Yaskawa INFORM job: SKRZYNIA_4840_0_STOPNI_1OBR.JBI

/JOB
//NAME SKRZYNIA_4840_0_STOPNI_1OBR
///FOLDERNAME 02-SKRZYNIE_JOBS
//POS
///NPOS 505,505,0,43,0,0
///TOOL 0
///POSTYPE PULSE
///PULSE
C00000=1055,-24125,84372,288,19725,204
C00001=1055,-24125,84372,288,19725,204
C00002=0,-15438,65714,0,-68532,0
C00003=25524,-25821,36823,19654,-58495,38520
C00004=23988,-24960,37134,18595,-57837,38812
C00005=22822,-23954,37534,17811,-57199,39017
C00006=22935,-24057,37491,17887,-57262,38997
C00007=20006,-24258,37408,15644,-56932,39751
C00008=24402,-25289,37013,18874,-58060,38740
C00009=22585,-24665,40358,17164,-59622,30036
C00010=23477,-23257,40205,18030,-58646,29630
C00011=22519,-22398,40568,17384,-58125,29795
C00012=22700,-22567,40495,17506,-58225,29764
C00013=19339,-22794,40398,14955,-57865,30607
C00014=24825,-24328,39798,18931,-59350,29401
C00015=32755,-32613,25711,29640,-48730,33694
C00016=25632,-30899,26166,23992,-46203,35378
C00017=24264,-29862,26497,22996,-45413,35639
C00018=24403,-29974,26459,23097,-45496,35612
C00019=20575,-30233,26374,19602,-44891,36810
C00020=26556,-31526,25988,24663,-46720,35206
C00021=30467,-39837,7164,47016,-28378,22959
C00022=27667,-31817,21023,40298,-29340,25942
C00023=26226,-30681,21430,39338,-28403,26129
C00024=26403,-30829,21375,39455,-28520,26106
C00025=23300,-31093,21277,35654,-27590,27434
C00026=27667,-31817,21023,40298,-29340,25942
C00027=26028,-43665,26580,-39946,8682,24640
C00028=27956,-30595,53065,-101898,6609,54413
C00029=26028,-43663,26580,-39944,8677,24639
C00030=38124,-35330,25507,26155,-45940,34419
C00031=17528,-33021,25719,14295,-44761,40001
C00032=28412,-21339,35361,20830,-70681,36412
C00033=27333,-20260,35973,20228,-70115,36596
C00034=27560,-20497,35837,20355,-70235,36556
C00035=24830,-20816,35654,18694,-69859,37222
C00036=28877,-18893,40191,20941,-72149,36569
C00037=27817,-32566,25782,25532,-47502,36865
C00038=25779,-31294,26110,24054,-46400,37243
C00039=24344,-30243,26427,23007,-45578,37515
C00040=24432,-30312,26405,23072,-45630,37498
C00041=20021,-30599,26315,19050,-44944,38872
C00042=26262,-31616,26021,24405,-46667,37153
C00043=27439,-32346,25835,25259,-47302,36935
C00044=25659,-31170,26146,23974,-46312,37260
C00045=24581,-30384,26384,23190,-45695,37464
C00046=24689,-30466,26358,23269,-45758,37444
C00047=20001,-30771,26264,18999,-45026,38899
C00048=26308,-31607,26026,24448,-46671,37139
C00049=29920,-29398,24569,49034,-27892,27689
C00050=29115,-28721,24834,48649,-27358,27707
C00051=27674,-27540,25333,47889,-26423,27783
C00052=27794,-27645,25287,47952,-26502,27777
C00053=24751,-27949,25156,44290,-25406,29014
C00054=29115,-28721,24834,48649,-27358,27707
C00055=46709,-36638,22429,58955,-37174,26391
C00056=28781,-29734,22128,31822,13650,18140
C00057=28781,-29734,22128,31822,47214,18140
C00058=28781,-29734,22128,31822,47214,18140
C00059=54276,-43673,-470,62120,-47739,23626
C00060=41752,-40945,238,55421,-40682,25053
C00061=39867,-39951,547,54583,-39468,25162
C00062=39963,-40004,529,54625,-39531,25157
C00063=37168,-40414,400,52318,-38319,25966
C00064=43368,-42081,-2849,57747,-40820,23950
C00065=38095,-40136,7813,41252,-44156,24924
C00066=33231,-38681,8176,37792,-41757,25918
C00067=31538,-37640,8473,36716,-40716,26179
C00068=31687,-37737,8444,36811,-40809,26155
C00069=27389,-38154,8322,32773,-39589,27627
C00070=33834,-39023,8084,38175,-42120,25821
C00071=27585,-47842,-289,32095,-40789,28095
C00072=4801,-35772,25187,4593,-28023,-82032
C00073=17634,-23800,39238,9573,-31425,-73339
C00074=17634,-23800,39238,9573,-31425,-73339
C00075=16549,-22464,39800,8390,-30730,-72975
C00076=16684,-22641,39722,8536,-30818,-73021
C00077=16684,-19968,45512,8078,-32771,-72767
C00078=17634,-23800,39238,9573,-31425,-73339
C00079=17837,-21535,44509,9322,-33342,-73155
C00080=17837,-21535,44509,9322,-33342,-73155
C00081=16866,-20378,45014,8305,-32755,-72853
C00082=17032,-20588,44918,8481,-32857,-72905
C00083=17032,-17542,51480,8009,-35060,-72636
C00084=17837,-21535,44509,9322,-33342,-73155
C00085=-20829,-18800,50532,-12466,-37179,-77446
C00086=-19934,-17904,50946,-11618,-36715,-77676
C00087=-20044,-18019,50891,-11723,-36773,-77647
C00088=-20044,-15288,56753,-11218,-38713,-77950
C00089=-20966,-18928,50473,-12596,-37250,-77413
C00090=-20884,-26676,33664,-14451,-31668,-76336
C00091=-20884,-26676,33664,-14451,-31668,-76336
C00092=-19557,-25338,34176,-13080,-30873,-76751
C00093=-19691,-25483,34117,-13220,-30955,-76709
C00094=-19691,-22773,39998,-12506,-32911,-77106
C00095=-20642,-26447,33747,-14206,-31526,-76411
C00096=-33629,-40566,17444,-29603,-33447,-71192
C00097=-33629,-40566,17444,42578,-32312,-84654
C00098=-42160,-31266,16400,42578,-32312,-84654
C00099=-87798,-804,48829,-20188,-26072,-60966
C00100=-76454,-11934,10236,-25964,7954,-64922
C00101=-76448,-11928,10235,-25961,7944,-64914
C00102=-68643,-7759,-23318,-14097,50582,-74897
C00103=-70868,-8793,-8075,-29663,30364,-70765
C00104=-67243,-1968,12282,-49553,26687,-63567
C00105=-68655,-309,14069,-48513,25966,-64203
C00106=-67497,-1678,12591,-49367,26558,-63682
C00107=-71436,-723,2905,-26484,35140,-73726
C00108=-71436,176,6426,-27636,33595,-73066
C00109=-71434,778,8668,-28412,32633,-72624
C00110=-68624,-2689,-85,-28291,36551,-72622
C00111=-99375,3692,5712,40719,48607,-84097
C00112=-94964,4957,10918,40408,44640,-83792
C00113=-93063,6047,12199,39572,43744,-83178
C00114=-94964,4957,10918,40408,44640,-83792
C00115=-94964,5754,13918,41385,43553,-84439
C00116=-94964,4957,10918,40408,44640,-83792
C00117=-90271,-412,-5146,23417,46876,-76529
C00118=-83133,-4088,-8267,6704,41492,-71542
C00119=-83133,-4088,-8267,6704,41492,-71542
C00120=-83133,-4088,-8267,6704,41492,-11598
C00121=-83133,-16026,-8267,6704,41492,-11598
C00122=-83133,-16026,-8267,6704,41492,-11598
C00123=-48225,-19387,30619,3889,32460,-6728
C00124=56943,-39861,25115,1795,-37402,-69601
C00125=29960,-38386,-19607,-115769,-41858,-24264
C00126=65721,-6478,18155,-133323,-22195,3361
C00127=70544,4411,32968,-134868,-18623,4660
C00128=71874,8263,38598,-134556,-17327,4659
C00129=72629,9390,40002,-135279,-16924,5107
C00130=71441,7638,37831,-134139,-17555,4406
C00131=77146,8888,25050,-166574,-32612,18372
C00132=77146,10029,28643,-166204,-31014,18167
C00133=77146,11198,32202,-165803,-29459,17947
C00134=75508,4678,16951,-165715,-35157,17778
C00135=68680,12216,24468,-164340,-40455,-13359
C00136=68362,12845,25743,-164045,-40097,-13561
C00137=68362,13700,28585,-163752,-38808,-13742
C00138=68362,12845,25743,-164045,-40097,-13561
C00139=64993,-1168,28876,-102971,-10760,-49875
C00140=63888,481,30670,-102324,-11438,-50313
C00141=64993,-1168,28876,-102971,-10760,-49875
C00142=58588,-14653,4620,-120782,-19611,-35794
C00143=29960,-38386,-19607,-115769,-41858,-24264
C00144=56943,-39861,25115,1795,-37402,-69601
C00145=-1002,-39861,25115,1795,-37402,-69601
C00146=-1001,-39858,25114,1795,-37402,0
C00147=6591,-33902,35532,5956,-1761,-1932
C00148=6592,-33900,35531,103508,-35512,-26314
C00149=-99253,-13690,44082,59847,13407,-31313
C00150=-85045,-36869,-4353,28502,-22832,-52282
C00151=-92346,-18713,13565,21110,-22545,-55257
C00152=-85732,-21202,11427,30682,-24763,-59235
C00153=-84559,-15616,15722,33768,-24118,-60665
C00154=-84150,-13282,17685,34842,-23935,-61163
C00155=-83260,-12880,18034,36130,-24218,-61709
C00156=-84150,-13282,17685,34842,-23935,-61163
C00157=-85365,-11775,19006,33430,-23307,-60600
C00158=-84150,-13282,17685,34842,-23935,-61163
C00159=-85786,-16909,14677,31743,-23900,-59790
C00160=-84150,-13282,17685,34842,-23935,-61163
C00161=-83215,-12861,18051,36194,-24233,-61735
C00162=-84150,-13282,17685,34842,-23935,-61163
C00163=-85327,-11825,18959,33476,-23327,-60618
C00164=-84150,-13282,17685,34842,-23935,-61163
C00165=-87841,-18519,13420,28367,-23534,-58339
C00166=-84150,-13282,17685,34842,-23935,-61163
C00167=-83292,-12894,18020,36083,-24208,-61688
C00168=-84150,-13282,17685,34842,-23935,-61163
C00169=-85185,-12008,18799,33646,-23400,-60687
C00170=-84150,-13282,17685,34842,-23935,-61163
C00171=-86371,-18277,13606,30568,-23951,-59265
C00172=-84345,-13370,17612,34554,-23873,-61041
C00173=-83240,-12871,18042,36158,-24225,-61720
C00174=-84345,-13370,17612,34554,-23873,-61041
C00175=-85365,-12110,18711,33368,-23345,-60568
C00176=-84345,-13370,17612,34554,-23873,-61041
C00177=-86191,-19647,12567,30467,-24278,-59187
C00178=-84345,-13372,17610,34552,-23873,-61039
C00179=-83096,-12807,18098,36363,-24268,-61804
C00180=-84345,-13372,17610,34552,-23873,-61039
C00181=-85268,-12232,18600,33480,-23393,-60612
C00182=-84345,-13372,17610,34552,-23873,-61039
C00183=-84814,-16043,15376,33312,-24093,-60464
C00184=-84104,-13265,17702,34906,-23948,-61189
C00185=-82960,-12743,18153,36555,-24313,-61887
C00186=-84104,-13265,17702,34906,-23948,-61189
C00187=-84979,-12194,18635,33901,-23496,-60788
C00188=-84104,-13265,17702,34906,-23948,-61189
C00189=-86610,-16845,14732,30573,-23614,-59301
C00190=-84104,-13265,17702,34906,-23948,-61189
C00191=-82793,-12667,18222,36790,-24370,-61986
C00192=-84104,-13265,17702,34906,-23948,-61189
C00193=-84888,-12305,18537,34004,-23540,-60830
C00194=-84104,-13265,17702,34906,-23948,-61189
C00195=-83806,-19585,12613,33764,-25080,-60559
C00196=-83675,-13072,17868,35530,-24083,-61453
C00197=-82553,-12556,18319,37130,-24451,-62127
C00198=-83675,-13072,17868,35530,-24083,-61453
C00199=-84378,-12223,18610,34735,-23716,-61138
C00200=-83675,-13072,17868,35530,-24083,-61453
C00201=-87149,-17993,13826,29513,-23647,-58830
C00202=-84104,-13265,17702,34906,-23948,-61189
C00203=-82640,-12594,18285,37014,-24425,-62079
C00204=-84104,-13265,17702,34906,-23948,-61189
C00205=-84792,-12429,18430,34119,-23592,-60877
C00206=-84104,-13265,17702,34906,-23948,-61189
C00207=-83583,-9185,30892,23668,-36042,-57025
C00208=-85789,-8328,35795,20592,-37093,-55378
C00209=-85786,-16735,14816,31782,-23869,-59812
C00210=-84103,-13263,17702,34906,-23947,-61191
C00211=-83225,-12865,18046,36177,-24227,-61729
C00212=-84103,-13263,17702,34906,-23947,-61191
C00213=-84774,-12447,18412,34138,-23599,-60886
C00214=-84103,-13263,17702,34906,-23947,-61191
C00215=-86149,-16246,6730,18897,-35239,-57128
C00216=-86244,-15289,7532,18875,-35060,-57127
C00217=-85361,-14893,7870,19824,-35193,-57574
C00218=-86244,-15289,7532,18875,-35060,-57127
C00219=-86889,-14409,8282,18264,-34784,-56850
C00220=-86244,-15289,7532,18875,-35060,-57127
C00221=-90262,-21765,2389,14114,-35574,-54847
C00222=-90262,-21765,2389,28730,-17672,-54847
C00223=-89967,-19086,25635,28730,-17672,-54847
C00224=568,-24029,84339,168,19981,112
C00225=568,-24677,83015,164,20405,113
C00226=101153,-24598,83176,165,20353,113
C00227=101153,-24598,83176,165,20353,113
C00228=89967,-19086,25635,-28730,-17672,54847
C00229=90262,-21765,2389,-28730,-17672,54847
C00230=86932,-18662,4771,-17876,-35519,56628
C00231=86578,-15436,7408,-18515,-35011,56957
C00232=85428,-14922,7844,-19753,-35183,57541
C00233=84405,-14447,8250,-20842,-35348,58054
C00234=85428,-14922,7844,-19753,-35183,57541
C00235=86134,-13973,8661,-19091,-34881,57237
C00236=85428,-14922,7844,-19753,-35183,57541
C00237=85786,-16735,14816,-31782,-23869,59812
C00238=83514,-12996,17929,-35760,-24132,61552
C00239=82296,-12429,18424,-37488,-24534,62281
C00240=83514,-12996,17929,-35760,-24132,61552
C00241=84266,-12085,18725,-34910,-23738,61214
C00242=83514,-12996,17929,-35760,-24132,61552
C00243=87323,-6914,39851,-18853,-38149,44508
C00244=83118,-12818,18089,-36330,-24263,61791
C00245=81969,-12276,18566,-37944,-24648,62472
C00246=83118,-12818,18089,-36330,-24263,61791
C00247=83927,-11846,18941,-35423,-23842,61433
C00248=83118,-12818,18089,-36330,-24263,61791
C00249=83806,-19585,12613,-33764,-25080,60559
C00250=83148,-12832,18077,-36287,-24254,61773
C00251=81889,-12236,18598,-38058,-24676,62520
C00252=83148,-12832,18077,-36287,-24254,61773
C00253=83900,-11930,18867,-35446,-23862,61440
C00254=83148,-12832,18077,-36287,-24254,61773
C00255=86610,-16845,14732,-30573,-23614,59301
C00256=82493,-13239,17725,-37070,-24559,62089
C00257=81442,-12739,18159,-38529,-24915,62703
C00258=82493,-13239,17725,-37070,-24559,62089
C00259=83435,-12133,18689,-36040,-24063,61682
C00260=82493,-13239,17725,-37070,-24559,62089
C00261=84814,-16043,15376,-33312,-24093,60464
C00262=82555,-13613,17404,-36910,-24580,62015
C00263=81369,-13053,17885,-38558,-24979,62709
C00264=82555,-13613,17404,-36910,-24580,62015
C00265=83568,-12431,18429,-35805,-24046,61580
C00266=82555,-13613,17404,-36910,-24580,62015
C00267=86191,-19647,12567,-30467,-24278,59187
C00268=82500,-13648,17375,-36975,-24607,62039
C00269=81594,-13224,17740,-38236,-24911,62571
C00270=82500,-13648,17375,-36975,-24607,62039
C00271=83449,-12543,18332,-35941,-24104,61633
C00272=82500,-13648,17375,-36975,-24607,62039
C00273=86371,-18277,13606,-30568,-23951,59265
C00274=82904,-13790,17251,-36416,-24470,61808
C00275=81796,-13275,17692,-37971,-24838,62464
C00276=82904,-13790,17251,-36416,-24470,61808
C00277=83696,-12867,18046,-35547,-24051,61466
C00278=82904,-13790,17251,-36416,-24470,61808
C00279=87841,-18519,13420,-28367,-23534,58339
C00280=82748,-13879,17174,-36603,-24542,61883
C00281=81789,-13434,17554,-37946,-24861,62449
C00282=82748,-13879,17174,-36603,-24542,61883
C00283=83603,-12888,18026,-35668,-24086,61514
C00284=82748,-13879,17174,-36603,-24542,61883
C00285=85786,-16909,14677,-31743,-23900,59790
C00286=82339,-14116,16972,-37087,-24733,62079
C00287=81557,-13752,17280,-38171,-24994,62536
C00288=82339,-14116,16972,-37087,-24733,62079
C00289=83390,-12909,18006,-35951,-24172,61633
C00290=82339,-14116,16972,-37087,-24733,62079
C00291=85732,-21202,11427,-30682,-24763,59235
C00292=82398,-14365,16763,-36952,-24745,62014
C00293=81340,-13876,17176,-38416,-25096,62632
C00294=82398,-14365,16763,-36952,-24745,62014
C00295=83629,-12951,17972,-35620,-24090,61491
C00296=82398,-14365,16763,-36952,-24745,62014
C00297=83775,-36460,5778,-32556,-23750,56951
C00298=69856,-53931,-13446,-33557,-28911,29591
C00299=0,-24029,84339,0,19981,0
C00300=0,-24029,84339,0,19981,0
C00301=0,-52280,40443,0,6876,0
C00302=43695,-41610,22646,45477,-37580,9181
C00303=79833,-32060,29151,65065,-75499,17030
C00304=46589,-23543,32575,47437,-59456,19719
C00305=35046,-28601,21000,31995,-60106,26294
C00306=20995,-31929,9410,15929,-60729,34224
C00307=58029,-25484,23838,55879,-68285,17494
C00308=64424,-28491,31029,58630,-66351,17656
C00309=0,-52280,40443,0,6876,0
C00310=0,-52280,40443,0,6876,0
C00311=23755,-47704,18289,26329,-25233,13971
C00312=32804,-46073,6525,41905,-31120,14425
C00313=62562,-39100,6547,70046,-55853,12125
C00314=48126,-33841,8393,64372,-47199,12361
C00315=31253,-44096,-7366,36514,-42480,22085
C00316=59828,-44646,-5405,72855,-48572,12139
C00317=0,-38761,66314,0,-763,0
C00318=0,-44757,54667,0,2744,0
C00319=40382,-38226,12225,48505,-40693,16039
C00320=55481,-27484,23768,62968,-54833,11978
C00321=49931,-26522,24223,59987,-51967,12537
C00322=41382,-34078,10932,46059,-50502,16311
C00323=55330,-33748,11238,57660,-59334,12681
C00324=78664,-24436,10378,82837,-79111,12029
C00325=75189,-23065,11287,81851,-76948,11927
C00326=75189,-45249,11287,81851,-38847,11927
C00327=29880,-45249,11287,43145,-11324,11927
C00328=0,-24029,84339,0,19981,0
C00329=0,-24026,84338,1,19977,2
C00330=4264,-34194,25387,4006,-26954,-29436
C00331=4264,-34194,25387,4006,-26954,-81856
C00332=-21478,-27798,32214,-15234,-31599,-76056
C00333=-19679,-23059,39354,-12567,-32689,-77067
C00334=16724,-20576,44291,8212,-32395,-72836
C00335=21329,-26386,39716,13285,-34016,-74401
C00336=-23778,-26243,38799,-16502,-35132,-75964
C00337=-20075,-15782,55752,-11329,-38404,-77896
C00338=16874,-17447,51356,7863,-34895,-72604
C00339=18580,-28601,30698,11472,-29284,-74138
C00340=6126,-41331,18955,6697,-26557,-30383
C00341=1,-24024,84337,2,19973,1
C00342=-64243,-26178,31107,-39513,40312,-5844
C00343=-72148,3973,56008,-35470,42045,-10522
C00344=-72090,16396,76301,-42067,35650,-6519
C00345=-69388,15725,61378,-31740,35177,-8719
C00346=-69127,27099,75569,-32744,34250,-8088
C00347=-67573,2495,11285,-21767,57629,-15193
C00348=-77819,19629,29798,-10454,63174,-20704
C00349=-72990,23583,14304,-10735,77209,-20379
C00350=-74593,38003,46707,-11043,65751,-19814
C00351=-73236,38943,48295,-11400,65557,-19316
C00352=-73329,42107,51779,-6346,67443,-19636
C00353=-87142,34654,46174,17622,63862,-25393
C00354=-87240,36727,48611,18897,66604,-25032
C00355=-99033,21517,12213,24947,79702,-26203
C00356=-91500,-14196,-34781,24472,81625,-22832
C00357=-100472,-45007,-27818,8167,67201,-29302
C00358=0,-36642,16905,0,48372,0
C00359=66009,-61997,-62105,21406,63483,18379
C00360=97242,-23579,-39442,10179,68876,30321
C00361=73684,-7073,-17511,24638,68131,29022
C00362=59136,7235,6676,33270,66602,27507
C00363=54816,14937,6234,39741,69494,31070
C00364=54365,20668,19279,41017,66202,29418
C00365=64503,4223,2857,29650,48528,26647
C00366=75622,3202,-3149,3890,49494,34281
C00367=88036,13177,2413,-18568,66573,35876
C00368=90462,21593,10123,-22613,76266,34479
C00369=92450,29224,20002,-25750,81642,33727
C00370=94949,8131,-12163,-20291,74229,36861
C00371=94949,8084,-13484,-20215,75047,36712
C00372=70412,-34016,-52305,-11724,65624,29757
C00373=44268,-30306,-1568,-7370,48673,18708
C00374=1,-24024,84337,2,19973,1
C00375=1,-24024,84337,2,19973,1
C00376=3796,-57671,22373,2336,-25309,-753
C00377=52632,-34554,16626,51161,-63050,5622
C00378=41454,-25301,37199,36495,-58855,24340
C00379=36675,-26014,30916,36565,-54296,30358
C00380=27394,-45680,-17645,86603,-20054,2054
C00381=62932,-33588,12189,66848,-61063,18031
C00382=55769,-31640,17107,64026,-54372,11197
C00383=49968,-26926,23568,59773,-52215,12586
C00384=49609,-31413,12230,55051,-55993,13121
C00385=55330,-33748,11238,57660,-59334,12681
C00386=29694,-28537,50295,31543,-18263,8508
C00387=1,-24024,84337,2,19973,1
C00388=1,-24024,84337,2,19973,1
C00389=57188,-41777,19973,48132,-58706,4905
C00390=55566,-48748,-16991,79805,-45048,-6941
C00391=49908,-48716,-25784,90749,-41340,-3650
C00392=34097,-50090,-26426,85195,-27377,-3312
C00393=25337,-51401,-46092,139691,-32480,-30357
C00394=55456,-69347,-61742,105381,-46819,-11205
C00395=12119,-24859,71505,13236,4440,2633
C00396=-91085,-34291,10385,1908,-24348,-42097
C00397=-86191,-19647,12567,30467,-24278,-59187
C00398=-99336,-11722,19052,-14323,-20229,-40037
C00399=-98356,-11562,19564,-10422,-20330,-41507
C00400=-99474,-20389,12397,-11593,-22150,-41069
C00401=0,-52280,40443,0,6876,0
C00402=98750,-34911,19055,13387,-20552,33529
C00403=85481,-22689,10385,-30594,-25183,59147
C00404=97204,-12655,18233,8807,-19987,42423
C00405=97248,-12883,18033,8874,-20029,42393
C00406=96230,-24528,9149,6144,-22576,43630
C00407=0,-52280,40443,0,6876,0
C00408=0,-52280,40443,0,6876,0
C00409=-90140,-60305,18108,-2708,1721,-7625
C00410=-95594,-27428,6866,-4663,-19832,-42154
C00411=-99356,-13410,18355,-15385,-17730,-37479
C00412=-99591,-10931,20459,-16242,-17374,-37088
C00413=-99412,-10883,20509,-15863,-17339,-37249
C00414=-100555,-16348,15834,-17428,-18409,-36628
C00415=-90140,-60305,18108,-2708,1721,-7625
C00416=0,-52280,40443,0,6876,0
C00417=84259,-57935,27522,-3761,3673,6310
C00418=86507,-39672,4297,-27618,-16640,46340
C00419=79502,-31038,5321,-35142,-29552,60614
C00420=87509,-17632,14108,-29072,-23467,58651
C00421=100494,-12641,18246,19637,-20925,37756
C00422=99867,-15453,10402,24266,-14765,33998
C00423=100699,-20865,6123,24471,-16015,33991
C00424=86507,-39672,4297,-27618,-16640,46340
C00425=84259,-57935,27522,-3761,3673,6310
C00426=0,-52280,40443,0,6876,0
C00427=0,-27933,77061,0,20812,0
C00428=0,-27933,77061,0,20812,0
C00429=0,-52280,40443,0,6876,0
C00430=-91970,-60791,14435,-3343,512,-9412
C00431=-99196,-15868,16098,-13748,-19297,-38710
C00432=-99196,-15868,16098,-13748,-19297,-38710
C00433=-99196,-15868,16098,-13748,-19297,-38710
C00434=-85896,-11794,19566,31613,-21074,-58206
C00435=-87494,-11929,19445,26784,-20178,-56163
C00436=-99562,-16264,15781,-14410,-19427,-38431
C00437=-99196,-15868,16098,-13748,-19297,-38710
C00438=-91970,-60791,14435,-3343,512,-9412
C00439=0,-52280,40443,0,6876,0
C00440=91083,-60784,14823,-9043,-825,15173
C00441=83869,-19403,12921,-33769,-24740,60260
C00442=83869,-19403,12921,-33769,-24740,60260
C00443=83420,-14897,16486,-35538,-24144,61113
C00444=90681,-11839,19658,-13770,-20778,51433
C00445=90505,-11641,19895,-14005,-20849,51502
C00446=95871,-14889,15992,4901,-19605,43825
C00447=83869,-19403,12921,-33769,-24740,60260
C00448=91083,-60784,14823,-9043,-825,15173
C00449=0,-52280,40443,0,6876,0
C00450=-91526,-60598,16699,7584,176,-13289
C00451=-94392,-6553,48683,5805,-47321,-49764
C00452=-88951,-345,54953,10686,-47392,-51569
C00453=-88305,5764,62037,11205,-47732,-51744
C00454=-91201,-14114,9416,8552,-34389,-51801
C00455=-84917,-15593,15742,33275,-23984,-60461
C00456=-81669,-15982,15425,37506,-25258,-62202
C00457=-79867,-25377,9541,37586,-25936,-59971
C00458=-91415,-60262,16631,7870,-73,-13734
C00459=24,-24029,84339,7,19981,5
C00460=160,-24029,84339,47,19981,32
C00461=99096,-24029,84339,47,19981,32
C00462=99096,-24029,84339,47,19981,32
C00463=89967,-19086,25635,-28730,-17672,54847
C00464=85786,-16735,14816,-31782,-23869,59812
C00465=83492,-14473,16674,-35480,-24338,61406
C00466=82747,-11488,19289,-37317,-24361,62210
C00467=85506,-13730,8787,-19466,-34817,57474
C00468=85505,-16299,6686,-19564,-35388,57437
C00469=89967,-19086,25635,-28730,-17672,54847
C00470=568,-24029,84339,168,19981,112
C00471=568,-24029,84339,168,19981,112
C00472=-91970,-60791,14435,-3343,512,-9412
C00473=-86948,-23217,10819,28314,-23349,-56438
C00474=-85895,-16522,15767,31843,-22281,-58087
C00475=-93744,1669,52928,2829,-38206,-34736
C00476=-93484,-766,47198,3260,-36104,-34933
C00477=-86145,-24679,9854,29028,-23971,-56682
C00478=-100471,-58311,4157,14142,-4822,-27614
C00479=-68517,-58311,4157,14142,-4822,-27614
C00480=0,-52280,40443,0,6876,0
C00481=91083,-60784,14823,-9043,-825,15173
C00482=83869,-19403,12921,-33769,-24740,60260
C00483=82620,-18743,14708,-32942,-26226,58979
C00484=84031,-4887,35984,-19530,-40379,54984
C00485=84316,-7987,27276,-19995,-38113,55712
C00486=84798,-22668,11879,-29033,-26372,57255
C00487=91083,-60784,14823,-9043,-825,15173
C00488=0,-52280,40443,0,6876,0
C00489=-6369,-39206,65423,-4801,-482,2563
C00490=-97287,-29142,12714,-8673,-22288,-37832
C00491=-86191,-19647,12567,30467,-24278,-59187
C00492=-85671,-16302,15857,30808,-24404,-58999
C00493=-100216,-10426,22391,-15020,-22581,-38655
C00494=-96259,-10424,22189,-2878,-17380,-43087
C00495=-87910,-17792,15835,25414,-24996,-56048
C00496=-97287,-29142,12714,-8673,-22288,-37832
C00497=0,-52280,40443,0,6876,0
C00498=92301,-25634,22749,2368,-15645,37646
C00499=83738,-18329,13570,-34202,-24868,60772
C00500=90255,-12942,18284,-15153,-20833,52586
C00501=93508,-13158,18002,-4292,-20124,47959
C00502=80226,-20465,12178,-39626,-27411,62762
C00503=92301,-25634,22749,2368,-15645,37646
C00504=0,-52280,40443,0,6876,0
BC00000=413138
BC00001=413138
BC00002=413138
BC00003=413134
BC00004=413134
BC00005=413134
BC00006=413134
BC00007=413134
BC00008=413134
BC00009=474623
BC00010=474628
BC00011=474628
BC00012=474628
BC00013=474628
BC00014=474628
BC00015=522849
BC00016=522849
BC00017=522849
BC00018=522849
BC00019=522849
BC00020=522849
BC00021=550624
BC00022=544410
BC00023=544410
BC00024=544410
BC00025=544410
BC00026=544410
BC00027=461029
BC00028=618860
BC00029=673957
BC00030=691345
BC00031=686969
BC00032=712250
BC00033=712250
BC00034=712250
BC00035=712250
BC00036=712250
BC00037=708270
BC00038=708270
BC00039=708270
BC00040=708270
BC00041=708270
BC00042=708270
BC00043=770184
BC00044=770184
BC00045=770184
BC00046=770184
BC00047=770184
BC00048=770184
BC00049=779519
BC00050=779519
BC00051=779519
BC00052=779519
BC00053=779519
BC00054=779519
BC00055=720678
BC00056=703565
BC00057=703565
BC00058=802913
BC00059=891475
BC00060=891475
BC00061=891475
BC00062=891475
BC00063=891475
BC00064=891475
BC00065=919114
BC00066=919114
BC00067=919114
BC00068=919114
BC00069=919114
BC00070=919114
BC00071=919114
BC00072=865069
BC00073=880430
BC00074=880430
BC00075=880430
BC00076=880430
BC00077=880430
BC00078=880430
BC00079=884876
BC00080=884876
BC00081=884876
BC00082=884876
BC00083=884876
BC00084=884876
BC00085=884876
BC00086=884876
BC00087=884876
BC00088=884876
BC00089=884876
BC00090=884876
BC00091=884876
BC00092=884876
BC00093=884876
BC00094=884876
BC00095=884876
BC00096=884876
BC00097=884876
BC00098=884876
BC00099=884876
BC00100=884876
BC00101=902628
BC00102=913714
BC00103=930418
BC00104=930418
BC00105=930418
BC00106=930418
BC00107=930418
BC00108=930418
BC00109=930419
BC00110=930419
BC00111=930419
BC00112=930419
BC00113=930419
BC00114=930419
BC00115=930419
BC00116=930419
BC00117=920796
BC00118=906162
BC00119=880897
BC00120=880897
BC00121=880897
BC00122=847715
BC00123=813282
BC00124=884876
BC00125=884876
BC00126=884876
BC00127=901090
BC00128=906251
BC00129=906251
BC00130=906251
BC00131=906251
BC00132=906251
BC00133=906251
BC00134=906251
BC00135=906251
BC00136=906251
BC00137=906251
BC00138=906251
BC00139=906251
BC00140=906251
BC00141=906251
BC00142=900738
BC00143=854154
BC00144=838793
BC00145=838793
BC00146=854156
BC00147=785093
BC00148=785096
BC00149=785096
BC00150=854699
BC00151=886829
BC00152=902188
BC00153=902188
BC00154=902188
BC00155=902188
BC00156=902188
BC00157=902188
BC00158=902188
BC00159=840744
BC00160=840744
BC00161=840744
BC00162=840744
BC00163=840744
BC00164=840744
BC00165=779300
BC00166=779300
BC00167=779300
BC00168=779300
BC00169=779300
BC00170=779300
BC00171=717855
BC00172=717855
BC00173=717855
BC00174=717855
BC00175=717855
BC00176=717855
BC00177=656405
BC00178=656405
BC00179=656405
BC00180=656405
BC00181=656405
BC00182=656405
BC00183=594961
BC00184=594961
BC00185=594961
BC00186=594961
BC00187=594961
BC00188=594961
BC00189=533517
BC00190=533517
BC00191=533517
BC00192=533517
BC00193=533517
BC00194=533517
BC00195=472073
BC00196=472073
BC00197=472073
BC00198=472073
BC00199=472073
BC00200=472073
BC00201=410629
BC00202=410629
BC00203=410629
BC00204=410629
BC00205=410629
BC00206=410629
BC00207=410629
BC00208=349186
BC00209=349186
BC00210=349186
BC00211=349186
BC00212=349186
BC00213=349186
BC00214=349186
BC00215=336469
BC00216=336469
BC00217=336469
BC00218=336469
BC00219=336469
BC00220=336469
BC00221=336469
BC00222=336469
BC00223=336469
BC00224=336469
BC00225=511557
BC00226=512005
BC00227=363797
BC00228=336469
BC00229=336469
BC00230=337415
BC00231=337415
BC00232=337415
BC00233=337415
BC00234=337415
BC00235=337415
BC00236=337415
BC00237=349186
BC00238=350137
BC00239=350137
BC00240=350137
BC00241=350137
BC00242=350137
BC00243=410629
BC00244=411580
BC00245=411580
BC00246=411580
BC00247=411580
BC00248=411580
BC00249=472073
BC00250=473025
BC00251=473025
BC00252=473025
BC00253=473025
BC00254=473025
BC00255=533517
BC00256=534468
BC00257=534468
BC00258=534468
BC00259=534468
BC00260=534468
BC00261=594961
BC00262=594961
BC00263=594961
BC00264=594961
BC00265=594961
BC00266=594961
BC00267=656405
BC00268=657350
BC00269=657350
BC00270=657350
BC00271=657350
BC00272=657350
BC00273=717855
BC00274=718799
BC00275=718799
BC00276=718799
BC00277=718799
BC00278=718799
BC00279=779300
BC00280=780245
BC00281=780245
BC00282=780245
BC00283=780245
BC00284=780245
BC00285=840744
BC00286=841691
BC00287=841691
BC00288=841691
BC00289=841691
BC00290=841691
BC00291=902188
BC00292=903136
BC00293=903136
BC00294=903136
BC00295=903136
BC00296=903136
BC00297=866428
BC00298=742376
BC00299=673191
BC00300=769966
BC00301=716865
BC00302=723595
BC00303=717171
BC00304=717171
BC00305=716481
BC00306=715784
BC00307=716000
BC00308=727625
BC00309=716865
BC00310=820009
BC00311=882789
BC00312=908954
BC00313=917484
BC00314=918947
BC00315=923719
BC00316=887066
BC00317=801718
BC00318=476098
BC00319=466373
BC00320=456696
BC00321=456696
BC00322=417276
BC00323=417276
BC00324=493986
BC00325=514306
BC00326=485368
BC00327=469222
BC00328=459569
BC00329=774064
BC00330=862181
BC00331=867397
BC00332=884876
BC00333=884876
BC00334=880429
BC00335=874663
BC00336=870174
BC00337=884876
BC00338=884876
BC00339=884104
BC00340=887696
BC00341=735557
BC00342=750919
BC00343=750919
BC00344=807629
BC00345=827515
BC00346=852454
BC00347=884386
BC00348=884386
BC00349=911895
BC00350=911895
BC00351=911895
BC00352=911896
BC00353=911896
BC00354=911897
BC00355=911897
BC00356=911897
BC00357=826555
BC00358=785153
BC00359=868693
BC00360=907813
BC00361=907814
BC00362=907814
BC00363=938061
BC00364=938061
BC00365=938061
BC00366=938061
BC00367=938061
BC00368=938064
BC00369=938064
BC00370=938064
BC00371=911658
BC00372=911658
BC00373=842845
BC00374=735557
BC00375=469153
BC00376=499904
BC00377=541592
BC00378=531564
BC00379=529848
BC00380=571759
BC00381=529848
BC00382=333808
BC00383=332068
BC00384=295166
BC00385=294388
BC00386=454783
BC00387=441730
BC00388=632615
BC00389=778314
BC00390=778312
BC00391=778312
BC00392=778312
BC00393=826760
BC00394=836556
BC00395=566410
BC00396=707357
BC00397=656405
BC00398=656405
BC00399=717855
BC00400=717855
BC00401=680147
BC00402=662303
BC00403=657350
BC00404=657350
BC00405=718803
BC00406=718803
BC00407=683493
BC00408=792672
BC00409=792672
BC00410=896850
BC00411=895720
BC00412=895720
BC00413=925351
BC00414=927080
BC00415=792672
BC00416=792672
BC00417=792672
BC00418=887446
BC00419=903126
BC00420=903126
BC00421=903126
BC00422=936389
BC00423=936389
BC00424=887446
BC00425=792672
BC00426=792672
BC00427=700249
BC00428=546214
BC00429=546214
BC00430=546211
BC00431=546211
BC00432=406776
BC00433=406776
BC00434=406778
BC00435=468200
BC00436=468200
BC00437=546211
BC00438=546211
BC00439=546214
BC00440=546214
BC00441=507604
BC00442=410782
BC00443=410782
BC00444=410782
BC00445=472720
BC00446=472720
BC00447=507604
BC00448=546214
BC00449=546214
BC00450=516757
BC00451=383716
BC00452=349186
BC00453=349186
BC00454=336469
BC00455=349186
BC00456=410629
BC00457=416512
BC00458=515801
BC00459=520018
BC00460=474013
BC00461=474013
BC00462=403108
BC00463=336469
BC00464=349186
BC00465=349186
BC00466=349186
BC00467=337415
BC00468=337415
BC00469=336469
BC00470=336469
BC00471=428401
BC00472=546211
BC00473=591088
BC00474=591088
BC00475=591088
BC00476=531116
BC00477=529640
BC00478=529640
BC00479=529640
BC00480=529640
BC00481=546214
BC00482=589919
BC00483=595627
BC00484=609761
BC00485=555903
BC00486=534177
BC00487=546214
BC00488=529640
BC00489=651195
BC00490=765890
BC00491=777968
BC00492=778453
BC00493=779252
BC00494=832733
BC00495=840748
BC00496=730002
BC00497=671551
BC00498=714120
BC00499=780224
BC00500=780222
BC00501=841743
BC00502=841743
BC00503=741100
BC00504=660586
///POSTYPE BASE
///RECTAN
///RCONF 1,0,0,0,0,0,0,0,0,0,0,0,0,0,0,0,0,0,0,0,0,0,0,0
P00006=0.000,0.000,0.000,0.0000,0.0000,0.0000
///RCONF 0,0,0,0,0,0,0,0,0,0,0,0,0,0,0,0,0,0,0,0,0,0,0,0
P00021=6.550,-0.003,-5.735,0.0000,0.0000,0.0000
P00022=5.943,-0.018,-6.388,0.0000,0.0000,0.0000
P00023=7.025,-0.019,-7.168,0.0000,0.0000,0.0000
P00024=5.926,-0.047,-4.777,0.0000,0.0000,0.0000
///RCONF 1,0,0,0,0,0,0,0,0,0,0,0,0,0,0,0,0,0,0,0,0,0,0,0
P00098=-0.089,-2.467,4.059,0.0000,0.0000,0.0000
P00099=0.011,-2.380,1.226,0.0000,0.0000,0.0000
P00100=-0.081,2.558,4.482,0.0000,0.0000,0.0000
P00101=0.030,-2.286,2.993,0.0000,0.0000,0.0000
P00102=-0.005,-1.108,1.644,0.0000,0.0000,0.0000
P00103=-0.094,-3.400,4.200,0.0000,0.0000,0.0000
P00104=0.043,-2.127,5.826,0.0000,0.0000,0.0000
P00105=-0.043,0.662,5.286,0.0000,0.0000,0.0000
P00106=-0.018,-2.519,0.237,0.0000,0.0000,0.0000
P00107=-0.008,-4.537,-4.500,0.0000,0.0000,0.0000
P00108=0.014,-3.040,2.637,0.0000,0.0000,0.0000
P00109=0.017,-3.622,2.341,0.0000,0.0000,0.0000
///RCONF 0,0,0,0,0,0,0,0,0,0,0,0,0,0,0,0,0,0,0,0,0,0,0,0
P00280=-0.761,-1.221,0.004,0.0000,0.0000,0.0000
///RCONF 1,0,0,0,0,0,0,0,0,0,0,0,0,0,0,0,0,0,0,0,0,0,0,0
P00281=-0.866,-3.587,-0.008,0.0000,0.0000,0.0000
///RCONF 0,0,0,0,1,0,0,0,0,0,0,0,0,0,0,0,0,0,0,0,0,0,0,0
P00290=-0.023,-0.050,5.560,0.0000,0.0000,0.0000
///RCONF 1,0,0,0,0,0,0,0,0,0,0,0,0,0,0,0,0,0,0,0,0,0,0,0
P00291=0.002,-0.893,4.526,0.0000,0.0000,0.0000
P00301=0.046,-2.112,7.779,0.0000,0.0000,0.0000
P00302=-0.180,-2.409,6.326,0.0000,0.0000,0.0000
///RCONF 0,0,0,0,0,0,0,0,0,0,0,0,0,0,0,0,0,0,0,0,0,0,0,0
P00303=-0.004,-1.437,-4.584,0.0000,0.0000,0.0000
P00304=0.028,-1.666,-4.234,0.0000,0.0000,0.0000
P00305=-0.003,-1.920,-3.501,0.0000,0.0000,0.0000
P00306=0.015,-2.252,-3.054,0.0000,0.0000,0.0000
P00307=0.019,-2.151,-5.077,0.0000,0.0000,0.0000
P00308=-0.003,-2.092,-4.888,0.0000,0.0000,0.0000
P00309=-0.040,-2.205,-4.992,0.0000,0.0000,0.0000
P00310=-0.006,-2.490,-5.925,0.0000,0.0000,0.0000
P00311=-0.007,-2.079,-5.307,0.0000,0.0000,0.0000
P00350=11.519,-0.008,1.149,0.0000,0.0000,0.0000
P00351=13.563,-0.027,-0.653,0.0000,0.0000,0.0000
P00352=13.252,-0.027,-0.827,0.0000,0.0000,0.0000
P00353=10.971,-0.082,0.776,0.0000,0.0000,0.0000
P00354=-0.024,2.508,-1.824,0.0000,0.0000,0.0000
P00355=-0.001,2.528,-1.131,0.0000,0.0000,0.0000
P00356=-0.034,2.921,-0.262,0.0000,0.0000,0.0000
P00357=0.003,3.386,-0.091,0.0000,0.0000,0.0000
P00358=0.014,3.037,-0.020,0.0000,0.0000,0.0000
P00359=-0.005,2.731,0.912,0.0000,0.0000,0.0000
P00360=-0.011,3.412,0.438,0.0000,0.0000,0.0000
//INST
///DATE 2025/06/04 08:15
///ATTR SC,RW
///GROUP1 RB1,BS1
NOP
CALL JOB:MOVE_INTO_TUNNEL
MOVJ C00000 BC00000 VJ=30.00
'------------------------
'------------------------
'SPOINA SRODEK DOL
'------------------------
'------------------------
'POMIAR DO WYJ!! PRZEROBIC NA STD
MOVJ C00001 BC00001 VJ=40.00
MOVJ C00002 BC00002 VJ=40.00
'W3P
MOVJ C00003 BC00003 VJ=20.00 PL=0
MOVL C00004 BC00004 V=166.7 PL=0
REFP 3 C00005 BC00005
CALL JOB:SEARCH-R1
SET P0100 P0006
SFTON P0100
MOVL C00006 BC00006 V=66.7 PL=0
REFP 3 C00007 BC00007
CALL JOB:SEARCH-R1
SET P0100 P0006
SFTON P0100
MOVL C00008 BC00008 V=333.3 PL=0
SFTOF
'W3L
MOVL C00009 BC00009 V=666.7
MOVL C00010 BC00010 V=166.7 PL=0
REFP 3 C00011 BC00011
CALL JOB:SEARCH-R1
SET P0101 P0006
SFTON P0101
MOVL C00012 BC00012 V=166.7 PL=0
REFP 3 C00013 BC00013
CALL JOB:SEARCH-R1
SET P0101 P0006
SFTON P0101
MOVL C00014 BC00014 V=333.3 PL=0
SFTOF
'W9P
MOVL C00015 BC00015 V=666.7
MOVL C00016 BC00016 V=166.7
REFP 3 C00017 BC00017
CALL JOB:SEARCH-R1
SET P0102 P0006
SFTON P0102
MOVL C00018 BC00018 V=166.7 PL=0
REFP 3 C00019 BC00019
CALL JOB:SEARCH-R1
SET P0102 P0006
SFTON P0102
SFTOF
MOVL C00020 BC00020 V=333.3 PL=0
'W9L
MOVL C00021 BC00021 V=666.7
MOVL C00022 BC00022 V=166.7
REFP 3 C00023 BC00023
CALL JOB:SEARCH-R1
SET P0103 P0006
SFTON P0103
MOVL C00024 BC00024 V=166.7 PL=0
REFP 3 C00025 BC00025
CALL JOB:SEARCH-R1
SET P0103 P0006
SFTON P0103
MOVL C00026 BC00026 V=333.3 PL=0
SFTOF
'PRZEJAZ NAD BELKA
MOVL C00027 BC00027 V=666.7
MOVJ C00028 BC00028 VJ=40.00
MOVJ C00029 BC00029 VJ=40.00
MOVJ C00030 BC00030 VJ=40.00
'W1P
SFTOF
MOVJ C00031 BC00031 VJ=20.00 PL=0
MOVL C00032 BC00032 V=166.7 PL=0
REFP 3 C00033 BC00033
CALL JOB:SEARCH-R1
SET P0104 P0006
SFTON P0104
MOVL C00034 BC00034 V=166.7 PL=0
REFP 3 C00035 BC00035
CALL JOB:SEARCH-R1
SET P0104 P0006
SFTON P0104
MOVL C00036 BC00036 V=333.3 PL=0
SFTOF
'W1L
MOVL C00037 BC00037 V=666.7
MOVL C00038 BC00038 V=166.7 PL=0
REFP 3 C00039 BC00039
CALL JOB:SEARCH-R1
SET P0105 P0006
SFTON P0105
MOVL C00040 BC00040 V=166.7 PL=0
REFP 3 C00041 BC00041
CALL JOB:SEARCH-R1
SET P0105 P0006
SFTON P0105
MOVL C00042 BC00042 V=333.3 PL=0
SFTOF
MOVL C00043 BC00043 V=666.7
'W10P
MOVL C00044 BC00044 V=166.7 PL=0
REFP 3 C00045 BC00045
CALL JOB:SEARCH-R1
SET P0106 P0006
SFTON P0106
MOVL C00046 BC00046 V=166.7 PL=0
REFP 3 C00047 BC00047
CALL JOB:SEARCH-R1
SET P0106 P0006
SFTON P0106
MOVL C00048 BC00048 V=333.3 PL=0
SFTOF
'W10L
MOVL C00049 BC00049 V=333.3
MOVL C00050 BC00050 V=166.7 PL=0
REFP 3 C00051 BC00051
CALL JOB:SEARCH-R1
SET P0107 P0006
SFTON P0107
MOVL C00052 BC00052 V=166.7 PL=0
REFP 3 C00053 BC00053
CALL JOB:SEARCH-R1
SET P0107 P0006
SFTON P0107
MOVL C00054 BC00054 V=333.3 PL=0
SFTOF
MOVL C00055 BC00055 V=333.3
MOVL C00056 BC00056 V=333.3
MOVL C00057 BC00057 V=333.3
MOVL C00058 BC00058 V=833.3
MOVL C00059 BC00059 V=333.3
MOVL C00060 BC00060 V=166.7 PL=0
REFP 3 C00061 BC00061
CALL JOB:SEARCH-R1
SET P0108 P0006
SFTON P0108
MOVL C00062 BC00062 V=166.7 PL=0
REFP 3 C00063 BC00063
CALL JOB:SEARCH-R1
SET P0108 P0006
SFTON P0108
MOVL C00064 BC00064 V=333.3 PL=0
SFTOF
'PRZEJAZD
MOVL C00065 BC00065 V=666.7
MOVL C00066 BC00066 V=166.7 PL=0
REFP 3 C00067 BC00067
CALL JOB:SEARCH-R1
SET P0109 P0006
SFTON P0109
MOVL C00068 BC00068 V=166.7 PL=0
REFP 3 C00069 BC00069
CALL JOB:SEARCH-R1
SET P0109 P0006
SFTON P0109
MOVL C00070 BC00070 V=333.3 PL=0
SFTOF
'PRZEJAZD
'POMIAR DO WYJ!! PRZEROBIC NA STD
'KONIEC
MOVJ C00071 BC00071 VJ=25.00
MOVJ C00072 BC00072 VJ=50.00
'W5L
MOVJ C00073 BC00073 VJ=30.00 PL=0
MOVL C00074 BC00074 V=166.7
REFP 3 C00075 BC00075
CALL JOB:SEARCH-R1
SET P0021 P0006
SFTON P0021
MOVL C00076 BC00076 V=166.7
REFP 3 C00077 BC00077
CALL JOB:SEARCH-R1
SET P0021 P0006
SFTON P0021
SFTOF
MOVL C00078 BC00078 V=166.7
'W6L
MOVJ C00079 BC00079 VJ=20.00 PL=0
MOVL C00080 BC00080 V=166.7
REFP 3 C00081 BC00081
CALL JOB:SEARCH-R1
SET P0022 P0006
SFTON P0022
MOVL C00082 BC00082 V=166.7
REFP 3 C00083 BC00083
CALL JOB:SEARCH-R1
SET P0022 P0006
SFTON P0022
SFTOF
MOVL C00084 BC00084 V=166.7
'W6P
MOVL C00085 BC00085 V=333.3 PL=0
REFP 3 C00086 BC00086
CALL JOB:SEARCH-R1
SET P0023 P0006
SFTON P0023
MOVL C00087 BC00087 V=166.7
REFP 3 C00088 BC00088
CALL JOB:SEARCH-R1
SET P0023 P0006
SFTON P0023
SFTOF
MOVL C00089 BC00089 V=166.7
'W5P
MOVJ C00090 BC00090 VJ=20.00 PL=0
MOVL C00091 BC00091 V=166.7
REFP 3 C00092 BC00092
CALL JOB:SEARCH-R1
SET P0024 P0006
SFTON P0024
MOVL C00093 BC00093 V=166.7
REFP 3 C00094 BC00094
CALL JOB:SEARCH-R1
SET P0024 P0006
SFTON P0024
SFTOF
MOVL C00095 BC00095 V=166.7
'W7A
MOVJ C00096 BC00096 VJ=40.00
MOVJ C00097 BC00097 VJ=40.00
MOVJ C00098 BC00098 VJ=40.00
MOVJ C00099 BC00099 VJ=40.00
MOVJ C00100 BC00100 VJ=40.00
MOVJ C00101 BC00101 VJ=40.00
MOVJ C00102 BC00102 VJ=40.00
MOVJ C00103 BC00103 VJ=40.00
MOVL C00104 BC00104 V=250.0
REFP 3 C00105 BC00105
CALL JOB:SEARCH-R1
SET P0280 P0006
SFTON P0280
MOVL C00106 BC00106 V=166.7
MOVL C00107 BC00107 V=250.0
MOVL C00108 BC00108 V=166.7
REFP 3 C00109 BC00109
CALL JOB:SEARCH-R1
SET P0280 P0006
MOVL C00110 BC00110 V=166.7
SFTOF
MOVL C00111 BC00111 V=333.3
MOVL C00112 BC00112 V=166.7
REFP 3 C00113 BC00113
CALL JOB:SEARCH-R1
SET P0290 P0006
SFTON P0290
MOVL C00114 BC00114 V=166.7
REFP 3 C00115 BC00115
CALL JOB:SEARCH-R1
SET P0290 P0006
MOVL C00116 BC00116 V=166.7
'DOKONCZYC SEARCH
'DOKONCZYC SEARCH
MOVJ C00117 BC00117 VJ=20.00
SFTOF
MOVJ C00118 BC00118 VJ=30.00
MOVJ C00119 BC00119 VJ=40.00
MOVJ C00120 BC00120 VJ=40.00
MOVJ C00121 BC00121 VJ=40.00
MOVJ C00122 BC00122 VJ=40.00
MOVJ C00123 BC00123 VJ=50.00
'W7B
MOVJ C00124 BC00124 VJ=50.00
MOVJ C00125 BC00125 VJ=50.00
MOVJ C00126 BC00126 VJ=30.00
MOVJ C00127 BC00127 VJ=20.00
MOVL C00128 BC00128 V=166.7
REFP 3 C00129 BC00129
CALL JOB:SEARCH-R1
SET P0281 P0006
MOVL C00130 BC00130 V=166.7
SFTON P0281
MOVL C00131 BC00131 V=166.7
MOVL C00132 BC00132 V=166.7
REFP 3 C00133 BC00133
CALL JOB:SEARCH-R1
SET P0281 P0006
MOVJ C00134 BC00134 VJ=15.00
SFTOF
MOVJ C00135 BC00135 VJ=20.00
MOVL C00136 BC00136 V=166.7
REFP 3 C00137 BC00137
CALL JOB:SEARCH-R1
SET P0291 P0006
MOVL C00138 BC00138 V=166.7
MOVL C00139 BC00139 V=166.7
REFP 3 C00140 BC00140
CALL JOB:SEARCH-R1
SET P0291 P0006
MOVL C00141 BC00141 V=166.7
MOVJ C00142 BC00142 VJ=30.00
MOVJ C00143 BC00143 VJ=30.00
MOVJ C00144 BC00144 VJ=50.00
MOVJ C00145 BC00145 VJ=50.00
'------------------------
'------------------------
'PRAWA STRONA PROFIL GORA
'------------------------
'------------------------
MOVJ C00146 BC00146 VJ=50.00
MOVJ C00147 BC00147 VJ=50.00
MOVJ C00148 BC00148 VJ=50.00
MOVJ C00149 BC00149 VJ=20.00
MOVJ C00150 BC00150 VJ=50.00
'------------------------
'W14A L
'------------------------
SFTOF
MOVJ C00151 BC00151 VJ=50.00
'------------------------
'W14A P
'------------------------
SFTOF
MOVJ C00152 BC00152 VJ=50.00
MOVJ C00153 BC00153 VJ=50.00
MOVL C00154 BC00154 V=166.7 PL=0
REFP 3 C00155 BC00155
CALL JOB:SEARCH-R1
SET P0301 P0006
SFTON P0301
MOVL C00156 BC00156 V=166.7 PL=0
REFP 3 C00157 BC00157
CALL JOB:SEARCH-R1
SET P0301 P0006
SFTON P0301
MOVL C00158 BC00158 V=166.7 PL=0
SFTOF
'------------------------
'W19A L
'------------------------
SFTOF
MOVJ C00159 BC00159 VJ=50.00
MOVL C00160 BC00160 V=200.0 PL=0
REFP 3 C00161 BC00161
CALL JOB:SEARCH-R1
SET P0302 P0006
SFTON P0302
MOVL C00162 BC00162 V=166.7 PL=0
REFP 3 C00163 BC00163
CALL JOB:SEARCH-R1
SET P0302 P0006
SFTON P0302
MOVL C00164 BC00164 V=250.0 PL=0
SFTOF
'------------------------
'W19A P
'------------------------
SFTOF
MOVJ C00165 BC00165 VJ=50.00
MOVL C00166 BC00166 V=166.7 PL=0
REFP 3 C00167 BC00167
CALL JOB:SEARCH-R1
SET P0303 P0006
SFTON P0303
MOVL C00168 BC00168 V=166.7 PL=0
REFP 3 C00169 BC00169
CALL JOB:SEARCH-R1
SET P0303 P0006
SFTON P0303
MOVL C00170 BC00170 V=166.7 PL=0
SFTOF
'------------------------
'W13A L
'------------------------
SFTOF
MOVJ C00171 BC00171 VJ=50.00
MOVL C00172 BC00172 V=166.7 PL=0
REFP 3 C00173 BC00173
CALL JOB:SEARCH-R1
SET P0304 P0006
SFTON P0304
MOVL C00174 BC00174 V=166.7 PL=0
REFP 3 C00175 BC00175
CALL JOB:SEARCH-R1
SET P0304 P0006
SFTON P0304
MOVL C00176 BC00176 V=166.7 PL=0
SFTOF
'------------------------
'W13A P
'------------------------
SFTOF
MOVJ C00177 BC00177 VJ=50.00
MOVL C00178 BC00178 V=200.0 PL=0
REFP 3 C00179 BC00179
CALL JOB:SEARCH-R1
SET P0305 P0006
SFTON P0305
MOVL C00180 BC00180 V=166.7 PL=0
REFP 3 C00181 BC00181
CALL JOB:SEARCH-R1
SET P0305 P0006
SFTON P0305
MOVL C00182 BC00182 V=250.0 PL=0
SFTOF
'------------------------
'W18A L
'------------------------
SFTOF
MOVJ C00183 BC00183 VJ=50.00
MOVL C00184 BC00184 V=200.0 PL=0
REFP 3 C00185 BC00185
CALL JOB:SEARCH-R1
SET P0306 P0006
SFTON P0306
MOVL C00186 BC00186 V=166.7 PL=0
REFP 3 C00187 BC00187
CALL JOB:SEARCH-R1
SET P0306 P0006
SFTON P0306
MOVL C00188 BC00188 V=166.7 PL=0
SFTOF
'------------------------
'W18A P
'------------------------
SFTOF
MOVJ C00189 BC00189 VJ=50.00
MOVL C00190 BC00190 V=200.0 PL=0
REFP 3 C00191 BC00191
CALL JOB:SEARCH-R1
SET P0307 P0006
SFTON P0307
MOVL C00192 BC00192 V=166.7 PL=0
REFP 3 C00193 BC00193
CALL JOB:SEARCH-R1
SET P0307 P0006
SFTON P0307
MOVL C00194 BC00194 V=166.7 PL=0
SFTOF
'------------------------
'W15A L
'------------------------
SFTOF
MOVJ C00195 BC00195 VJ=50.00
MOVL C00196 BC00196 V=200.0 PL=0
REFP 3 C00197 BC00197
CALL JOB:SEARCH-R1
SET P0308 P0006
SFTON P0308
MOVL C00198 BC00198 V=166.7 PL=0
REFP 3 C00199 BC00199
CALL JOB:SEARCH-R1
SET P0308 P0006
SFTON P0308
MOVL C00200 BC00200 V=166.7 PL=0
SFTOF
'------------------------
'W15A P
'------------------------
SFTOF
MOVJ C00201 BC00201 VJ=50.00
MOVL C00202 BC00202 V=166.7 PL=0
REFP 3 C00203 BC00203
CALL JOB:SEARCH-R1
SET P0309 P0006
SFTON P0309
MOVL C00204 BC00204 V=166.7 PL=0
REFP 3 C00205 BC00205
CALL JOB:SEARCH-R1
SET P0309 P0006
SFTON P0309
MOVL C00206 BC00206 V=166.7 PL=0
SFTOF
MOVL C00207 BC00207 V=333.3
'------------------------
'W17A L
'------------------------
MOVL C00208 BC00208 V=500.0
SFTOF
MOVJ C00209 BC00209 VJ=20.00
MOVL C00210 BC00210 V=166.7 PL=0
REFP 3 C00211 BC00211
CALL JOB:SEARCH-R1
SET P0310 P0006
SFTON P0310
MOVL C00212 BC00212 V=166.7 PL=0
REFP 3 C00213 BC00213
CALL JOB:SEARCH-R1
SET P0310 P0006
SFTON P0310
MOVL C00214 BC00214 V=166.7 PL=0
SFTOF
'------------------------
'W17A P
'------------------------
SFTOF
MOVL C00215 BC00215 V=416.7
MOVL C00216 BC00216 V=166.7 PL=0
REFP 3 C00217 BC00217
CALL JOB:SEARCH-R1
SET P0311 P0006
SFTON P0311
MOVL C00218 BC00218 V=166.7 PL=0
REFP 3 C00219 BC00219
CALL JOB:SEARCH-R1
SET P0311 P0006
SFTON P0311
MOVL C00220 BC00220 V=166.7 PL=0
SFTOF
MOVJ C00221 BC00221 VJ=10.00
MOVJ C00222 BC00222 VJ=20.00
MOVJ C00223 BC00223 VJ=50.00
MOVJ C00224 BC00224 VJ=50.00
MOVJ C00225 BC00225 VJ=70.00
MOVJ C00226 BC00226 VJ=30.00
MOVJ C00227 BC00227 VJ=30.00
'------------------------
'------------------------
'LEWA STRONA PROFIL GORA
'------------------------
'------------------------
MOVJ C00228 BC00228 VJ=30.00
MOVJ C00229 BC00229 VJ=30.00
MOVJ C00230 BC00230 VJ=30.00
'------------------------
'W17B L
'------------------------
SFTOF
MOVJ C00231 BC00231 VJ=15.00
MOVL C00232 BC00232 V=166.7 PL=0
REFP 3 C00233 BC00233
CALL JOB:SEARCH-R1
SET P0350 P0006
SFTON P0350
MOVL C00234 BC00234 V=166.7 PL=0
REFP 3 C00235 BC00235
CALL JOB:SEARCH-R1
SET P0350 P0006
SFTON P0350
MOVL C00236 BC00236 V=166.7 PL=0
SFTOF
'------------------------
'W17B P
'------------------------
SFTOF
MOVL C00237 BC00237 V=333.3
MOVL C00238 BC00238 V=166.7 PL=0
REFP 3 C00239 BC00239
CALL JOB:SEARCH-R1
SET P0351 P0006
SFTON P0351
MOVL C00240 BC00240 V=166.7 PL=0
REFP 3 C00241 BC00241
CALL JOB:SEARCH-R1
SET P0351 P0006
SFTON P0351
MOVL C00242 BC00242 V=166.7 PL=0
SFTOF
'POPRAWID DOJAZD
'------------------------
'W15B L
'------------------------
SFTOF
MOVJ C00243 BC00243 VJ=10.00
MOVL C00244 BC00244 V=166.7 PL=0
REFP 3 C00245 BC00245
CALL JOB:SEARCH-R1
SET P0352 P0006
SFTON P0352
MOVL C00246 BC00246 V=166.7 PL=0
REFP 3 C00247 BC00247
CALL JOB:SEARCH-R1
SET P0352 P0006
SFTON P0352
MOVL C00248 BC00248 V=166.7 PL=0
SFTOF
'------------------------
'W15B P
'------------------------
SFTOF
MOVJ C00249 BC00249 VJ=20.00
MOVL C00250 BC00250 V=166.7 PL=0
REFP 3 C00251 BC00251
CALL JOB:SEARCH-R1
SET P0353 P0006
SFTON P0353
MOVL C00252 BC00252 V=166.7 PL=0
REFP 3 C00253 BC00253
CALL JOB:SEARCH-R1
SET P0353 P0006
SFTON P0353
MOVL C00254 BC00254 V=166.7 PL=0
SFTOF
'------------------------
'W18B L
'------------------------
SFTOF
MOVJ C00255 BC00255 VJ=50.00
MOVL C00256 BC00256 V=166.7 PL=0
REFP 3 C00257 BC00257
CALL JOB:SEARCH-R1
SET P0354 P0006
SFTON P0354
MOVL C00258 BC00258 V=166.7 PL=0
REFP 3 C00259 BC00259
CALL JOB:SEARCH-R1
SET P0354 P0006
SFTON P0354
MOVL C00260 BC00260 V=166.7 PL=0
SFTOF
'------------------------
'W18B P
'------------------------
SFTOF
MOVJ C00261 BC00261 VJ=50.00
MOVL C00262 BC00262 V=166.7 PL=0
REFP 3 C00263 BC00263
CALL JOB:SEARCH-R1
SET P0355 P0006
SFTON P0355
MOVL C00264 BC00264 V=166.7 PL=0
REFP 3 C00265 BC00265
CALL JOB:SEARCH-R1
SET P0355 P0006
SFTON P0355
MOVL C00266 BC00266 V=166.7 PL=0
SFTOF
'------------------------
'W13B L
'------------------------
SFTOF
MOVJ C00267 BC00267 VJ=50.00
MOVL C00268 BC00268 V=166.7 PL=0
REFP 3 C00269 BC00269
CALL JOB:SEARCH-R1
SET P0356 P0006
SFTON P0356
MOVL C00270 BC00270 V=166.7 PL=0
REFP 3 C00271 BC00271
CALL JOB:SEARCH-R1
SET P0356 P0006
SFTON P0356
MOVL C00272 BC00272 V=166.7 PL=0
SFTOF
'------------------------
'W13B P
'------------------------
SFTOF
MOVJ C00273 BC00273 VJ=50.00
MOVL C00274 BC00274 V=166.7 PL=0
REFP 3 C00275 BC00275
CALL JOB:SEARCH-R1
SET P0357 P0006
SFTON P0357
MOVL C00276 BC00276 V=166.7 PL=0
REFP 3 C00277 BC00277
CALL JOB:SEARCH-R1
SET P0357 P0006
SFTON P0357
MOVL C00278 BC00278 V=166.7 PL=0
SFTOF
'------------------------
'W19B L
'------------------------
SFTOF
MOVJ C00279 BC00279 VJ=50.00
MOVL C00280 BC00280 V=166.7 PL=0
REFP 3 C00281 BC00281
CALL JOB:SEARCH-R1
SET P0358 P0006
SFTON P0358
MOVL C00282 BC00282 V=166.7 PL=0
REFP 3 C00283 BC00283
CALL JOB:SEARCH-R1
SET P0358 P0006
SFTON P0358
MOVL C00284 BC00284 V=166.7 PL=0
SFTOF
'------------------------
'W19B P
'------------------------
SFTOF
MOVJ C00285 BC00285 VJ=50.00
MOVL C00286 BC00286 V=166.7 PL=0
REFP 3 C00287 BC00287
CALL JOB:SEARCH-R1
SET P0359 P0006
SFTON P0359
MOVL C00288 BC00288 V=166.7 PL=0
REFP 3 C00289 BC00289
CALL JOB:SEARCH-R1
SET P0359 P0006
SFTON P0359
MOVL C00290 BC00290 V=166.7 PL=0
SFTOF
'------------------------
'W14B L
'------------------------
SFTOF
MOVJ C00291 BC00291 VJ=50.00
MOVL C00292 BC00292 V=166.7 PL=0
REFP 3 C00293 BC00293
CALL JOB:SEARCH-R1
SET P0360 P0006
SFTON P0360
MOVL C00294 BC00294 V=166.7 PL=0
REFP 3 C00295 BC00295
CALL JOB:SEARCH-R1
SET P0360 P0006
SFTON P0360
MOVL C00296 BC00296 V=166.7 PL=0
SFTOF
'------------------------
'W14B P
'------------------------
SFTOF
SFTOF
MOVJ C00297 BC00297 VJ=50.00
MOVJ C00298 BC00298 VJ=50.00
MOVJ C00299 BC00299 VJ=50.00
'WELD
'WELD
'WELD
MOVJ C00300 BC00300 VJ=10.00
'**********************
'**********************
'POCZATEK SPAWANIA DOL
'**********************
'**********************
''
'**********************
'W1
'**********************
MOVJ C00301 BC00301 VJ=50.00
MOVJ C00302 BC00302 VJ=40.00
MOVL C00303 BC00303 V=166.7
SFTON P0105
MOVL C00304 BC00304 V=166.7
MACRO1 MJ#(0) ARGF24
ARCON
SFTON P0104
MOVL C00305 BC00305 V=11.3
MOVL C00306 BC00306 V=11.3
ARCOF
SFTOF
MOVL C00307 BC00307 V=333.3
MOVJ C00308 BC00308 VJ=20.00
MOVJ C00309 BC00309 VJ=30.00
MOVJ C00310 BC00310 VJ=50.00
MOVJ C00311 BC00311 VJ=40.00
MOVJ C00312 BC00312 VJ=20.00
'**********************
'W2
'**********************
MOVL C00313 BC00313 V=166.7
SFTON P0109
MOVL C00314 BC00314 V=333.3
ARCON
SFTON P0108
MOVL C00315 BC00315 V=10.8
ARCOF
SFTOF
MOVL C00316 BC00316 V=333.3
MOVJ C00317 BC00317 VJ=40.00
MOVJ C00318 BC00318 VJ=70.00
MOVJ C00319 BC00319 VJ=20.00
MOVL C00320 BC00320 V=666.7
'**********************
'W3
'**********************
SFTON P0101
MOVL C00321 BC00321 V=166.7
ARCON
SFTON P0100
MOVL C00322 BC00322 V=11.7
ARCOF
MOVL C00323 BC00323 V=166.7
SFTOF
MOVJ C00324 BC00324 VJ=30.00
MOVJ C00325 BC00325 VJ=30.00
MOVJ C00326 BC00326 VJ=50.00
MOVJ C00327 BC00327 VJ=30.00
MOVJ C00328 BC00328 VJ=40.00
'**********************
'W5
'**********************
MOVJ C00329 BC00329 VJ=50.00
COMM MOVJ C00330 BC00330 VJ=25.00
COMM MOVJ C00331 BC00331 VJ=30.00
COMM '**********************
COMM 'W5
COMM MOVL C00332 BC00332 V=333.3
COMM '**********************
COMM MACRO1 MJ#(0) ARGF9
COMM SFTON P0024
COMM MOVL C00333 BC00333 V=166.7
COMM ARCON
COMM SFTON P0021
COMM MOVL C00334 BC00334 V=10.8
COMM ARCOF
COMM SFTOF
COMM MOVJ C00335 BC00335 VJ=20.00
COMM MOVJ C00336 BC00336 VJ=20.00
COMM '**********************
COMM 'W6
COMM '**********************
COMM MACRO1 MJ#(0) ARGF9
COMM SFTON P0023
COMM MOVL C00337 BC00337 V=250.0
COMM ARCON
COMM SFTON P0022
COMM MOVL C00338 BC00338 V=10.8
COMM ARCOF
COMM SFTOF
COMM MOVJ C00339 BC00339 VJ=10.00
COMM MOVJ C00340 BC00340 VJ=30.00
MOVJ C00341 BC00341 VJ=40.00
MOVJ C00342 BC00342 VJ=40.00
MOVJ C00343 BC00343 VJ=40.00
MOVJ C00344 BC00344 VJ=40.00
MOVJ C00345 BC00345 VJ=20.00
MOVJ C00346 BC00346 VJ=10.00
MOVJ C00347 BC00347 VJ=20.00
MOVL C00348 BC00348 V=166.7
MACRO1 MJ#(0) ARGF14
MOVL C00349 BC00349 V=166.7
SFTON P0280
MOVL C00350 BC00350 V=166.7 PL=0
ARCON ASF#(22)
MOVL C00351 BC00351 V=9.2
MOVL C00352 BC00352 V=9.2
SFTON P0290
MOVL C00353 BC00353 V=9.2
MOVL C00354 BC00354 V=9.2
ARCOF
SFTOF
MOVL C00355 BC00355 V=250.0
MOVL C00356 BC00356 V=416.7
MOVJ C00357 BC00357 VJ=30.00
MOVJ C00358 BC00358 VJ=30.00
MOVJ C00359 BC00359 VJ=30.00
MOVJ C00360 BC00360 VJ=30.00
MOVJ C00361 BC00361 VJ=30.00
'7b
MOVL C00362 BC00362 V=333.3
MOVL C00363 BC00363 V=333.3
SFTON P0281
MOVL C00364 BC00364 V=166.7 PL=0
ARCON ASF#(22)
MOVL C00365 BC00365 V=9.2
MOVL C00366 BC00366 V=9.2
SFTON P0291
MOVL C00367 BC00367 V=9.2
MOVL C00368 BC00368 V=9.2
MOVL C00369 BC00369 V=9.2
ARCOF
SFTOF
'TUTAJ DODAC 7
'TUTAJ DODAC 7
'TUTAJ DODAC 7
MOVL C00370 BC00370 V=333.3
MOVL C00371 BC00371 V=333.3
MOVL C00372 BC00372 V=333.3
MOVJ C00373 BC00373 VJ=20.00
MOVJ C00374 BC00374 VJ=30.00
MOVJ C00375 BC00375 VJ=50.00
MOVJ C00376 BC00376 VJ=50.00
MOVJ C00377 BC00377 VJ=40.00
'**********************
'W9
'**********************
MACRO1 MJ#(0) ARGF24
MOVL C00378 BC00378 V=166.7
SFTON P0102
MOVL C00379 BC00379 V=166.7
ARCON
SFTON P0103
MOVL C00380 BC00380 V=11.3
ARCOF
SFTOF
MOVL C00381 BC00381 V=333.3
'**********************
'SPOINA_PODLOGA_BRAK_ROZP
'**********************
MOVL C00382 BC00382 V=333.3
SFTON P0099
MOVL C00383 BC00383 V=166.7
ARCON
SFTON P0098
MOVL C00384 BC00384 V=11.7
ARCOF
MOVL C00385 BC00385 V=166.7
SFTOF
'SPOINA_PODLOGA_BRAK_ROZP
MOVJ C00386 BC00386 VJ=25.00
MOVJ C00387 BC00387 VJ=40.00
MOVJ C00388 BC00388 VJ=70.00
MOVJ C00389 BC00389 VJ=50.00
MOVJ C00390 BC00390 VJ=20.00
'**********************
'W10
'**********************
MOVL C00391 BC00391 V=333.3
SFTON P0106
MOVL C00392 BC00392 V=166.7
ARCON
SFTON P0107
MOVL C00393 BC00393 V=11.3
ARCOF
SFTOF
MOVL C00394 BC00394 V=333.3
MOVJ C00395 BC00395 VJ=50.00
'**********************
'**********************
'POCZATEK SPAWANIA BOKI
'**********************
'**********************
MOVJ C00396 BC00396 VJ=50.00
MOVJ C00397 BC00397 VJ=50.00
'**********************
'W13A
'**********************
SFTON P0305
MOVL C00398 BC00398 V=250.0 PL=0
SFTOF
MACRO1 MJ#(0) ARGF10
ARCON
SFTON P0304
MOVL C00399 BC00399 V=10.8
ARCOF
SFTOF
MOVL C00400 BC00400 V=250.0
'W13B
MOVJ C00401 BC00401 VJ=30.00
MOVJ C00402 BC00402 VJ=50.00
MOVL C00403 BC00403 V=500.0
'**********************
'W13B
'**********************
SFTON P0356
MOVL C00404 BC00404 V=166.7 PL=0
SFTOF
ARCON
SFTON P0357
MOVL C00405 BC00405 V=10.8
ARCOF
SFTOF
MOVL C00406 BC00406 V=250.0
MOVJ C00407 BC00407 VJ=30.00
MOVJ C00408 BC00408 VJ=40.00
MOVJ C00409 BC00409 VJ=30.00
MOVJ C00410 BC00410 VJ=30.00
'**********************
'W14A
'**********************
MOVL C00411 BC00411 V=250.0
SFTON P0301
MOVL C00412 BC00412 V=133.3 PL=0
SFTOF
ARCON
SFTON P0301
MOVL C00413 BC00413 V=10.8
ARCOF
SFTOF
MOVL C00414 BC00414 V=150.0
MOVJ C00415 BC00415 VJ=40.00
MOVJ C00416 BC00416 VJ=30.00
MOVJ C00417 BC00417 VJ=30.00
MOVJ C00418 BC00418 VJ=30.00
MOVJ C00419 BC00419 VJ=30.00
'**********************
'W14B
'**********************
SFTON P0360
MOVL C00420 BC00420 V=333.3
MOVL C00421 BC00421 V=166.7 PL=0
ARCON
MOVL C00422 BC00422 V=10.8
ARCOF
SFTOF
MOVL C00423 BC00423 V=250.0
MOVJ C00424 BC00424 VJ=40.00
MOVJ C00425 BC00425 VJ=40.00
MOVJ C00426 BC00426 VJ=30.00
MOVJ C00427 BC00427 VJ=40.00
MOVJ C00428 BC00428 VJ=30.00
MOVJ C00429 BC00429 VJ=30.00
MOVJ C00430 BC00430 VJ=30.00
MOVJ C00431 BC00431 VJ=30.00
MOVJ C00432 BC00432 VJ=30.00
'**********************
'W15A
'**********************
SFTON P0309
MOVL C00433 BC00433 V=166.7
MOVL C00434 BC00434 V=166.7 PL=0
SFTOF
ARCON
SFTON P0308
MOVL C00435 BC00435 V=10.8
ARCOF
SFTOF
MOVL C00436 BC00436 V=150.0
MOVJ C00437 BC00437 VJ=30.00
MOVJ C00438 BC00438 VJ=50.00
MOVJ C00439 BC00439 VJ=50.00
MOVJ C00440 BC00440 VJ=50.00
MOVJ C00441 BC00441 VJ=50.00
MOVJ C00442 BC00442 VJ=50.00
'**********************
'W15B
'**********************
SFTON P0352
MOVL C00443 BC00443 V=250.0
MOVL C00444 BC00444 V=83.3 PL=0
SFTOF
ARCON
SFTON P0353
MOVL C00445 BC00445 V=10.8
ARCOF
MOVL C00446 BC00446 V=66.7
SFTOF
MOVJ C00447 BC00447 VJ=40.00
MOVJ C00448 BC00448 VJ=50.00
MOVJ C00449 BC00449 VJ=50.00
'BRAK W TEJ DLUGOSCI
'**********************
'W16A
'**********************
'**********************
'W16B
'**********************
'BRAK W TEJ DLUGOSCI
'**********************
'W17A
'**********************
MOVJ C00450 BC00450 VJ=50.00
MOVJ C00451 BC00451 VJ=50.00
'**********************
'W17A
'**********************
SFTON P0310
MOVL C00452 BC00452 V=333.3
MOVL C00453 BC00453 V=166.7 PL=0
SFTOF
ARCON
SFTON P0311
MOVL C00454 BC00454 V=10.8
ARCOF
SFTOF
MOVL C00455 BC00455 V=333.3
MOVJ C00456 BC00456 VJ=30.00
MOVJ C00457 BC00457 VJ=30.00
MOVJ C00458 BC00458 VJ=50.00
MOVJ C00459 BC00459 VJ=50.00
MOVJ C00460 BC00460 VJ=50.00
MOVJ C00461 BC00461 VJ=50.00
MOVJ C00462 BC00462 VJ=50.00
MOVJ C00463 BC00463 VJ=30.00
MOVJ C00464 BC00464 VJ=30.00
'**********************
'W17B
'**********************
SFTON P0351
MOVL C00465 BC00465 V=166.7
MOVL C00466 BC00466 V=166.7 PL=0
SFTOF
ARCON
SFTON P0350
MOVL C00467 BC00467 V=10.8
ARCOF
SFTOF
MOVL C00468 BC00468 V=250.0
MOVJ C00469 BC00469 VJ=30.00
MOVJ C00470 BC00470 VJ=30.00
MOVJ C00471 BC00471 VJ=30.00
MOVJ C00472 BC00472 VJ=30.00
MOVJ C00473 BC00473 VJ=40.00
'**********************
'W18A
'**********************
SFTON P0306
MOVL C00474 BC00474 V=333.3
MOVL C00475 BC00475 V=166.7 PL=0
SFTOF
ARCON
SFTON P0307
MOVL C00476 BC00476 V=10.8
ARCOF
SFTOF
MOVL C00477 BC00477 V=250.0
MOVJ C00478 BC00478 VJ=30.00
MOVJ C00479 BC00479 VJ=30.00
MOVJ C00480 BC00480 VJ=50.00
MOVJ C00481 BC00481 VJ=50.00
MOVJ C00482 BC00482 VJ=50.00
'**********************
'W18B
'**********************
SFTON P0355
MOVL C00483 BC00483 V=166.7
MOVL C00484 BC00484 V=166.7 PL=0
SFTOF
ARCON
SFTON P0354
MOVL C00485 BC00485 V=10.8
ARCOF
MOVL C00486 BC00486 V=250.0
SFTOF
MOVJ C00487 BC00487 VJ=30.00
MOVJ C00488 BC00488 VJ=30.00
MOVJ C00489 BC00489 VJ=40.00
MOVJ C00490 BC00490 VJ=50.00
MOVJ C00491 BC00491 VJ=30.00
'**********************
'W19A
'**********************
MOVL C00492 BC00492 V=166.7
SFTON P0303
MOVL C00493 BC00493 V=166.7 PL=0
SFTOF
ARCON
SFTON P0302
MOVL C00494 BC00494 V=10.8
ARCOF
SFTOF
MOVL C00495 BC00495 V=150.0
MOVJ C00496 BC00496 VJ=30.00
MOVJ C00497 BC00497 VJ=50.00
MOVJ C00498 BC00498 VJ=50.00
'**********************
'W19B
'**********************
SFTON P0358
MOVL C00499 BC00499 V=500.0
MOVL C00500 BC00500 V=166.7 PL=0
SFTOF
ARCON
SFTON P0359
MOVL C00501 BC00501 V=10.8
ARCOF
SFTOF
MOVL C00502 BC00502 V=250.0
MOVJ C00503 BC00503 VJ=40.00
MOVJ C00504 BC00504 VJ=50.00
CALL JOB:MOVE_OUT_OF_TUNNEL
END
